// Mitsubishi GX Works2 project: PLC_Group_12   PLC: FX3G

// global labels: Global1
VAR_GLOBAL
  start_day AT X010 : BOOL;
  flour_input AT D1100 : REAL;
  yeast_input AT D1102 : REAL;
  water_input AT D1104 : REAL;
  oil_input AT D1106 : REAL;
  spices_input AT D1108 : REAL;
  flour_stock AT D1110 : REAL;
  yeast_stock AT D1112 : REAL;
  water_stock AT D1114 : REAL;
  oil_stock AT D1116 : REAL;
  spices_stock AT D1118 : REAL;
  input AT M0 : BOOL;
END_VAR
VAR_GLOBAL CONSTANT
  min_flour : REAL := 100;
END_VAR
VAR_GLOBAL
  enough_flour AT M20 : BOOL;
  const1 AT E5.0 : REAL;
  const2 AT E2.0 : REAL;
  const4 AT E10.0 : REAL;
  const3 AT E0.3 : REAL;
  enough_yeast AT M40 : BOOL;
  enough_water AT M42 : BOOL;
  enough_oil AT M44 : BOOL;
  enough_spices AT M46 : BOOL;
  emergemcy_stop AT X007 : BOOL;
  all_ok AT M6 : BOOL;
  can_start AT M52 : BOOL;
  in_process AT Y010 : BOOL;
  flour_tank AT D1120 : REAL;
  yeast_tank AT D1122 : REAL;
  water_tank AT D1124 : REAL;
  oil_tank AT D1126 : REAL;
  spices_tank AT D1128 : REAL;
  start_prepare AT X002 : BOOL;
  sub_flour AT E100 : REAL;
  add_flour AT E100 : REAL;
  sub_yeast AT E20 : REAL;
  add_yeast AT E20 : REAL;
  sub_water AT E50 : REAL;
  add_water AT E50 : REAL;
  sub_oil AT E30 : REAL;
  add_oil AT E30 : REAL;
  sub_spices AT E10 : REAL;
  add_spices AT E10 : REAL;
  preparing_lamp AT Y005 : BOOL;
  preparing_timer AT TC200 : BOOL;
  timer_stopped AT TS200 : BOOL;
  start_mix AT X001 : BOOL;
  mix_tank AT D1130 : REAL;
  rst_flour AT E0.0 : REAL;
  rst_material AT E0.0 : REAL;
  mixTankActivaited AT M101 : BOOL;
  mixer_lamp AT Y001 : BOOL;
  start_swelling AT X011 : BOOL;
  counter_one AT CC0 : BOOL;
  swelling_tank AT D1132 : REAL;
  counter AT CS0 : BOOL;
  swellingProccesActivated AT M102 : BOOL;
  swelling_timer AT TC201 : BOOL;
  one_sec_pulse AT M8013 : BOOL;
  swelling_one AT Y002 : BOOL;
  swelling_two AT Y003 : BOOL;
  timer_two_stopped AT TS201 : BOOL;
  baking_procces_activated AT M103 : BOOL;
  baking_pan AT D1134 : REAL;
  baking_timer AT TC202 : BOOL;
  baking_lamp AT Y004 : BOOL;
  quality_ck AT X003 : BOOL;
  quality AT D8281 : INT;
  temp_analog_value AT D1200 : INT;
  quality_value AT D1202 : REAL;
  qc_approve AT M104 : BOOL;
  qc_fail_counter AT CC2 : BOOL;
  qc_timer AT TC203 : BOOL;
  qc_lamp AT Y006 : BOOL;
  shelves AT D1136 : REAL;
  QA_Activated AT M105 : BOOL;
  all_reset AT M340 : BOOL;
  not_enough_material AT M341 : BOOL;
  TC204 : BOOL;
  end_timer AT TC204 : BOOL;
  stop_acticated AT M350 : BOOL;
  emptyMix_Tank_checkPulse : BOOL;
  day_active_counter AT CC8 : BOOL;
  preperingLampIsOver AT M110 : BOOL;
  moveToTanksConfimation AT M100 : BOOL;
  bakingLampsOver AT M112 : BOOL;
  stopSystemTimerActivated AT M342 : BOOL;
  test AT M106 : BOOL;
  testtwo AT M107 : BOOL;
  qc_approval AT M108 : BOOL;
  testthree AT M109 : BOOL;
END_VAR

// task Task_01 (event TRUE, interval 0, priority 31): POU_01

PROGRAM POU_01
VAR
  day_active : BOOL;
END_VAR
(* structured ladder/FBD written out as ST: instructions are called as NAME(EN, inputs, outputs); _pN, _eN, _tN stand for wires *)
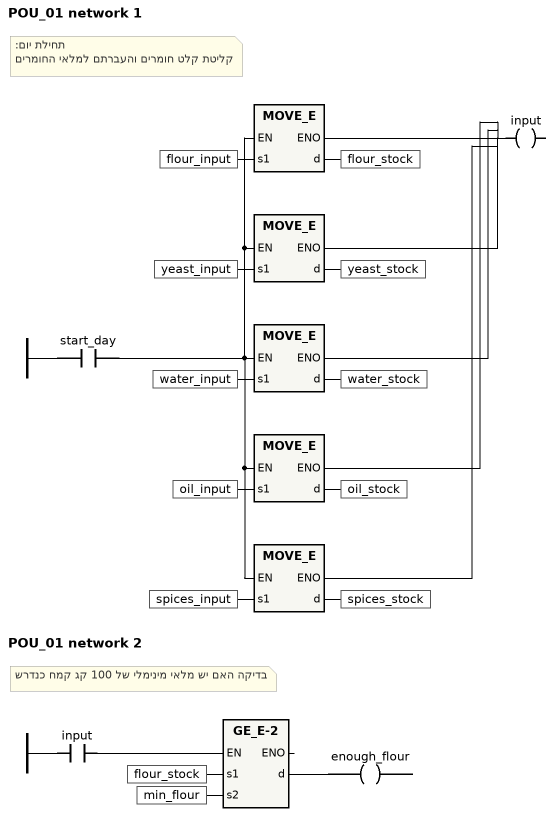
(* network 1 *)
(* תחילת יום: /  קליטת קלט חומרים והעברתם למלאי החומרים *)
_e1 := MOVE_E(start_day, flour_input, flour_stock);
_e2 := MOVE_E(start_day, yeast_input, yeast_stock);
_e3 := MOVE_E(start_day, water_input, water_stock);
_e4 := MOVE_E(start_day, oil_input, oil_stock);
_e5 := MOVE_E(start_day, spices_input, spices_stock);
input := _e1 OR _e2 OR _e3 OR _e4 OR _e5;
(* network 2 *)
(* בדיקה האם יש מלאי מינימלי של 100 קג קמח כנדרש *)
GE_E(input, flour_stock, min_flour, _t1);
enough_flour := _t1;
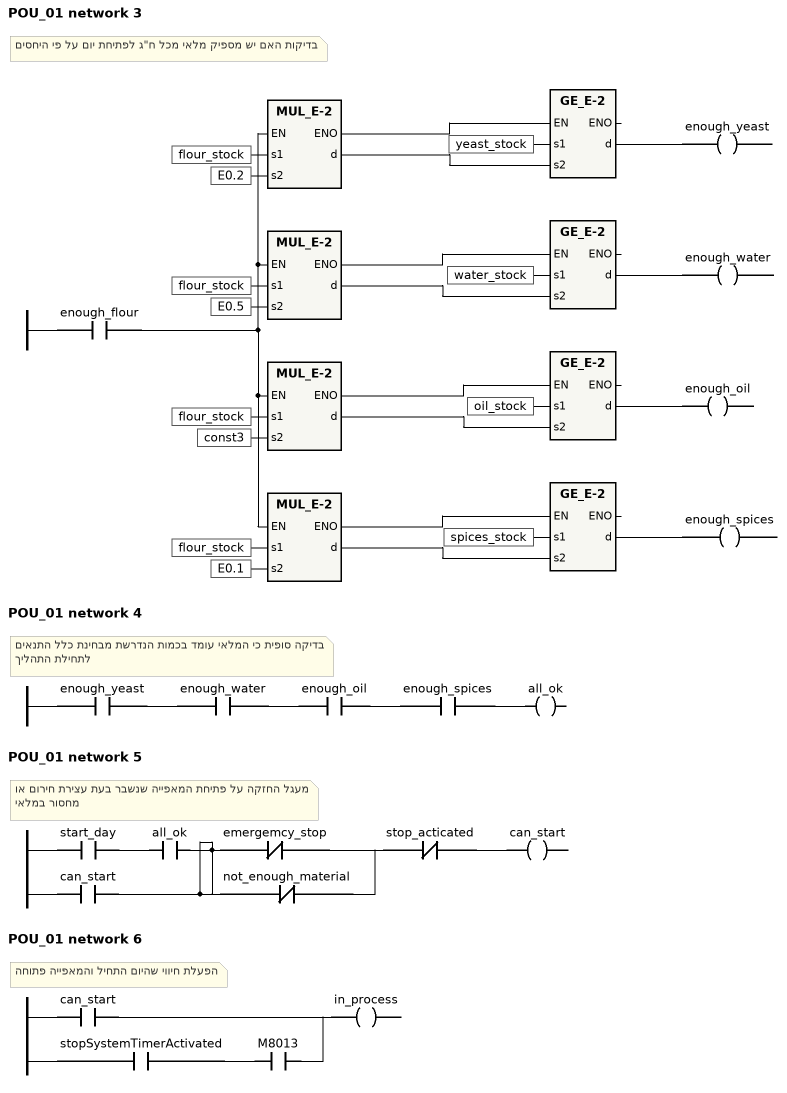
(* network 3 *)
(* בדיקות האם יש מספיק מלאי מכל ח"ג לפתיחת יום על פי היחסים *)
_e2 := MUL_E(enough_flour, flour_stock, E0.2, _t1);
GE_E(_e2, yeast_stock, _t1, _t3);
enough_yeast := _t3;
_e5 := MUL_E(enough_flour, flour_stock, E0.5, _t4);
GE_E(_e5, water_stock, _t4, _t6);
enough_water := _t6;
_e8 := MUL_E(enough_flour, flour_stock, const3, _t7);
GE_E(_e8, oil_stock, _t7, _t9);
enough_oil := _t9;
_e11 := MUL_E(enough_flour, flour_stock, E0.1, _t10);
GE_E(_e11, spices_stock, _t10, _t12);
enough_spices := _t12;
(* network 4 *)
(* בדיקה סופית כי המלאי עומד בכמות הנדרשת מבחינת כלל התנאים לתחילת התהליך *)
all_ok := enough_yeast AND enough_water AND enough_oil AND enough_spices;
(* network 5 *)
(* מעגל החזקה על פתיחת המאפייה שנשבר בעת עצירת חירום או מחסור במלאי *)
_p1 := (start_day AND all_ok) OR can_start;
can_start := ((_p1 AND NOT emergemcy_stop) OR (_p1 AND NOT not_enough_material)) AND NOT stop_acticated;
(* network 6 *)
(* הפעלת חיווי שהיום התחיל והמאפייה פתוחה *)
in_process := can_start OR (stopSystemTimerActivated AND M8013);
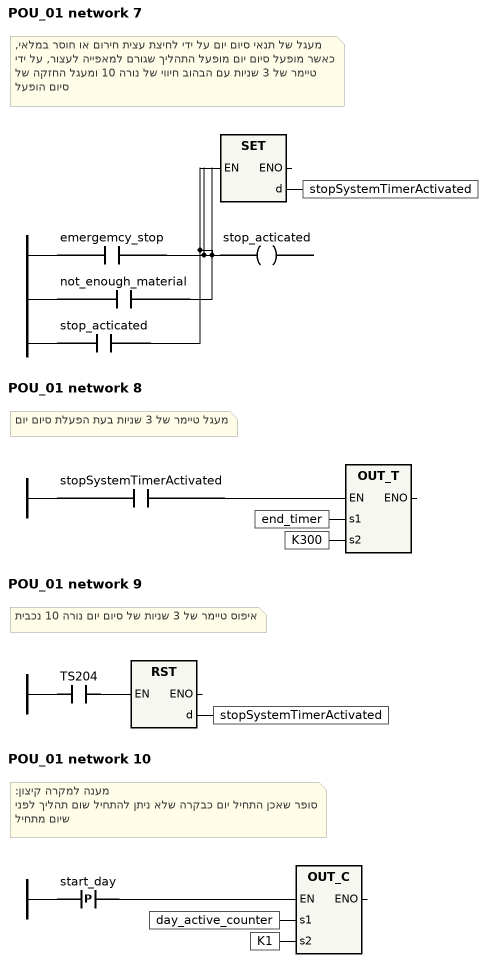
(* network 7 *)
(* מעגל של תנאי סיום יום על ידי לחיצת עצית חירום או חוסר במלאי, /  כאשר מופעל סיום יום מופעל התהליך שגורם למאפייה לעצור, על ידי טיימר של 3 שניות עם הבהוב חיווי של נורה 10 ומעגל החזקה של סיום הופעל *)
_p1 := emergemcy_stop OR not_enough_material OR stop_acticated;
SET(_p1, stopSystemTimerActivated);
stop_acticated := _p1;
(* network 8 *)
(* מעגל טיימר של 3 שניות בעת הפעלת סיום יום *)
OUT_T(stopSystemTimerActivated, end_timer, K300);
(* network 9 *)
(* איפוס טיימר של 3 שניות של סיום יום נורה 10 נכבית *)
RST(TS204, stopSystemTimerActivated);
(* network 10 *)
(* מענה למקרה קיצון: / סופר שאכן התחיל יום כבקרה שלא ניתן להתחיל שום תהליך לפני שיום מתחיל *)
OUT_C(LDP(TRUE, start_day), day_active_counter, K1);
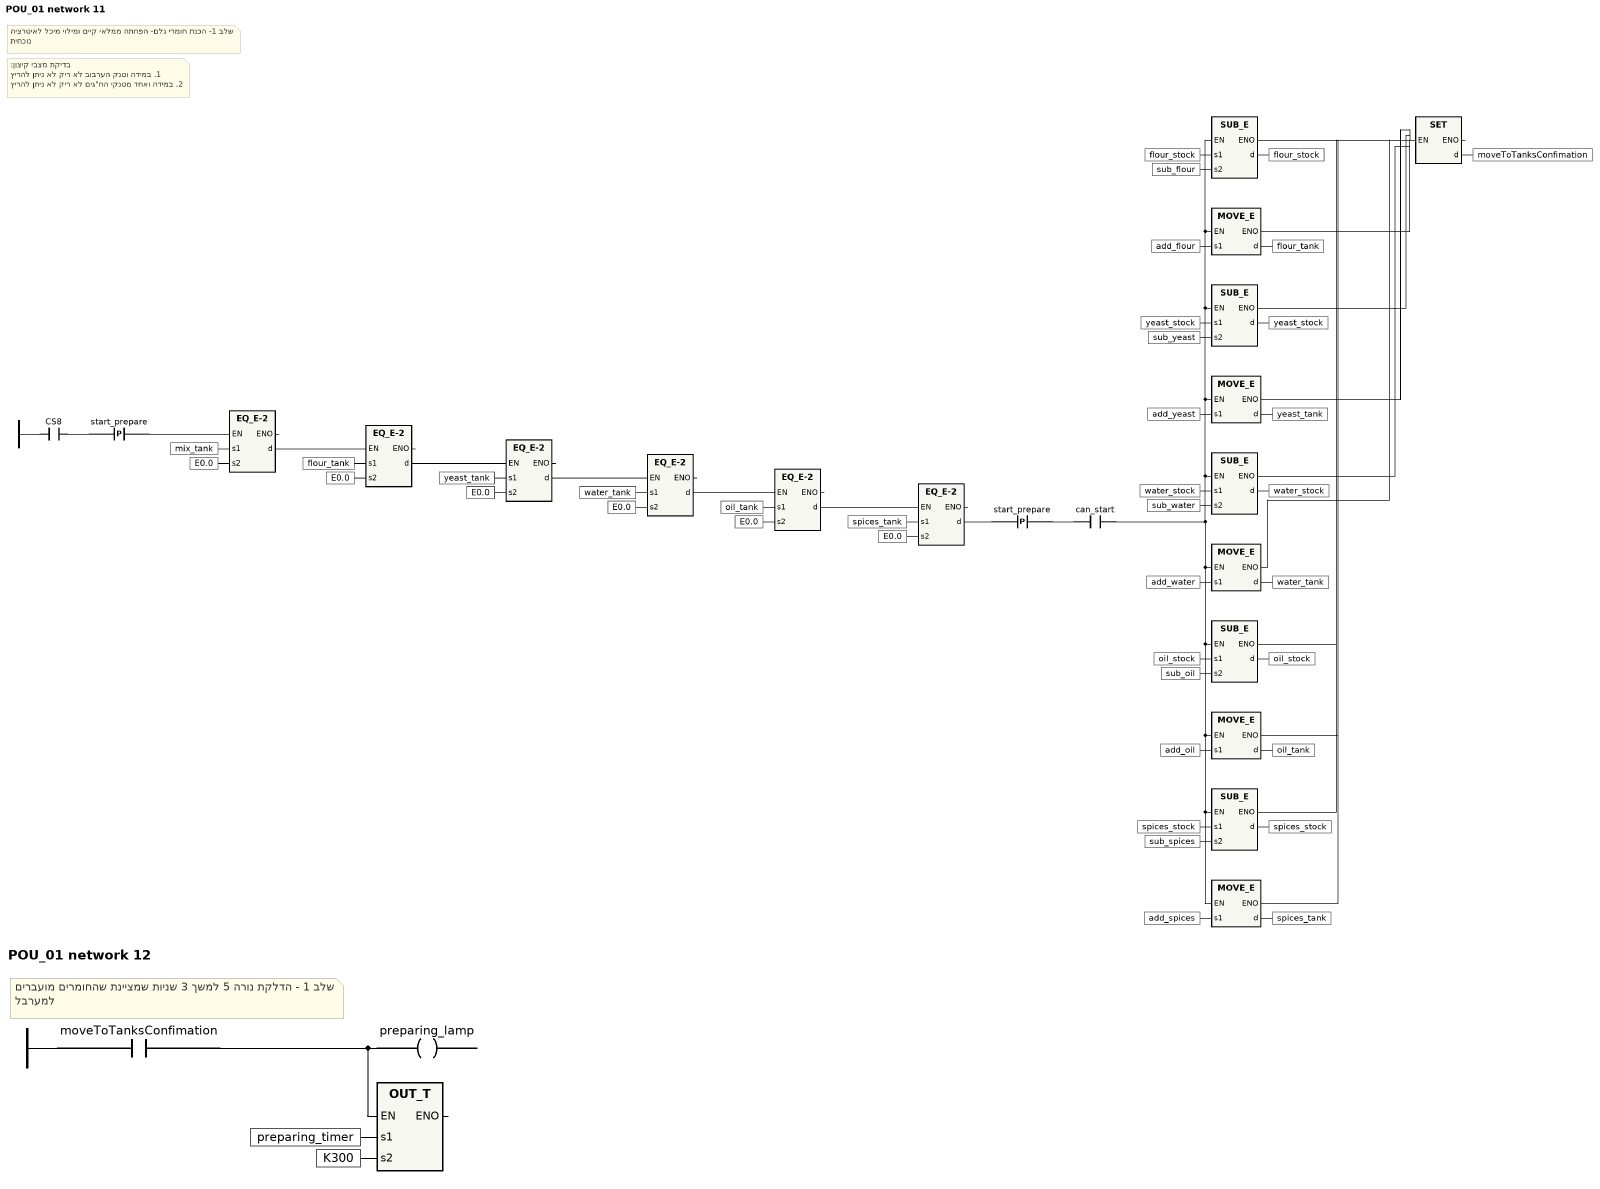
(* network 11 *)
(* שלב 1- הכנת חומרי גלם- הפחתה ממלאי קיים ומילוי מיכל לאיטרציה נוכחית *)
(* בדיקת מצבי קיצון: / 1. במידה וטנק הערבוב לא ריק לא ניתן להריץ / 2. במידה ואחד מטנקי הח"גים לא ריק לא ניתן להריץ *)
EQ_E(CS8 AND LDP(TRUE, start_prepare), mix_tank, E0.0, _t1);
EQ_E(_t1, flour_tank, E0.0, _t2);
EQ_E(_t2, yeast_tank, E0.0, _t3);
EQ_E(_t3, water_tank, E0.0, _t4);
EQ_E(_t4, oil_tank, E0.0, _t5);
EQ_E(_t5, spices_tank, E0.0, _t6);
_p7 := _t6 AND LDP(TRUE, start_prepare) AND can_start;
_e8 := SUB_E(_p7, flour_stock, sub_flour, flour_stock);
_e9 := MOVE_E(_p7, add_flour, flour_tank);
_e10 := SUB_E(_p7, yeast_stock, sub_yeast, yeast_stock);
_e11 := MOVE_E(_p7, add_yeast, yeast_tank);
_e12 := SUB_E(_p7, water_stock, sub_water, water_stock);
_e13 := MOVE_E(_p7, add_water, water_tank);
_e14 := SUB_E(_p7, oil_stock, sub_oil, oil_stock);
_e15 := MOVE_E(_p7, add_oil, oil_tank);
_e16 := SUB_E(_p7, spices_stock, sub_spices, spices_stock);
_e17 := MOVE_E(_p7, add_spices, spices_tank);
SET(_e8 OR _e9 OR _e10 OR _e11 OR _e12 OR _e13 OR _e14 OR _e15 OR _e16 OR _e17, moveToTanksConfimation);
(* network 12 *)
(* שלב 1 - הדלקת נורה 5 למשך 3 שניות שמציינת שהחומרים מועברים למערבל *)
preparing_lamp := moveToTanksConfimation;
OUT_T(moveToTanksConfimation, preparing_timer, K300);
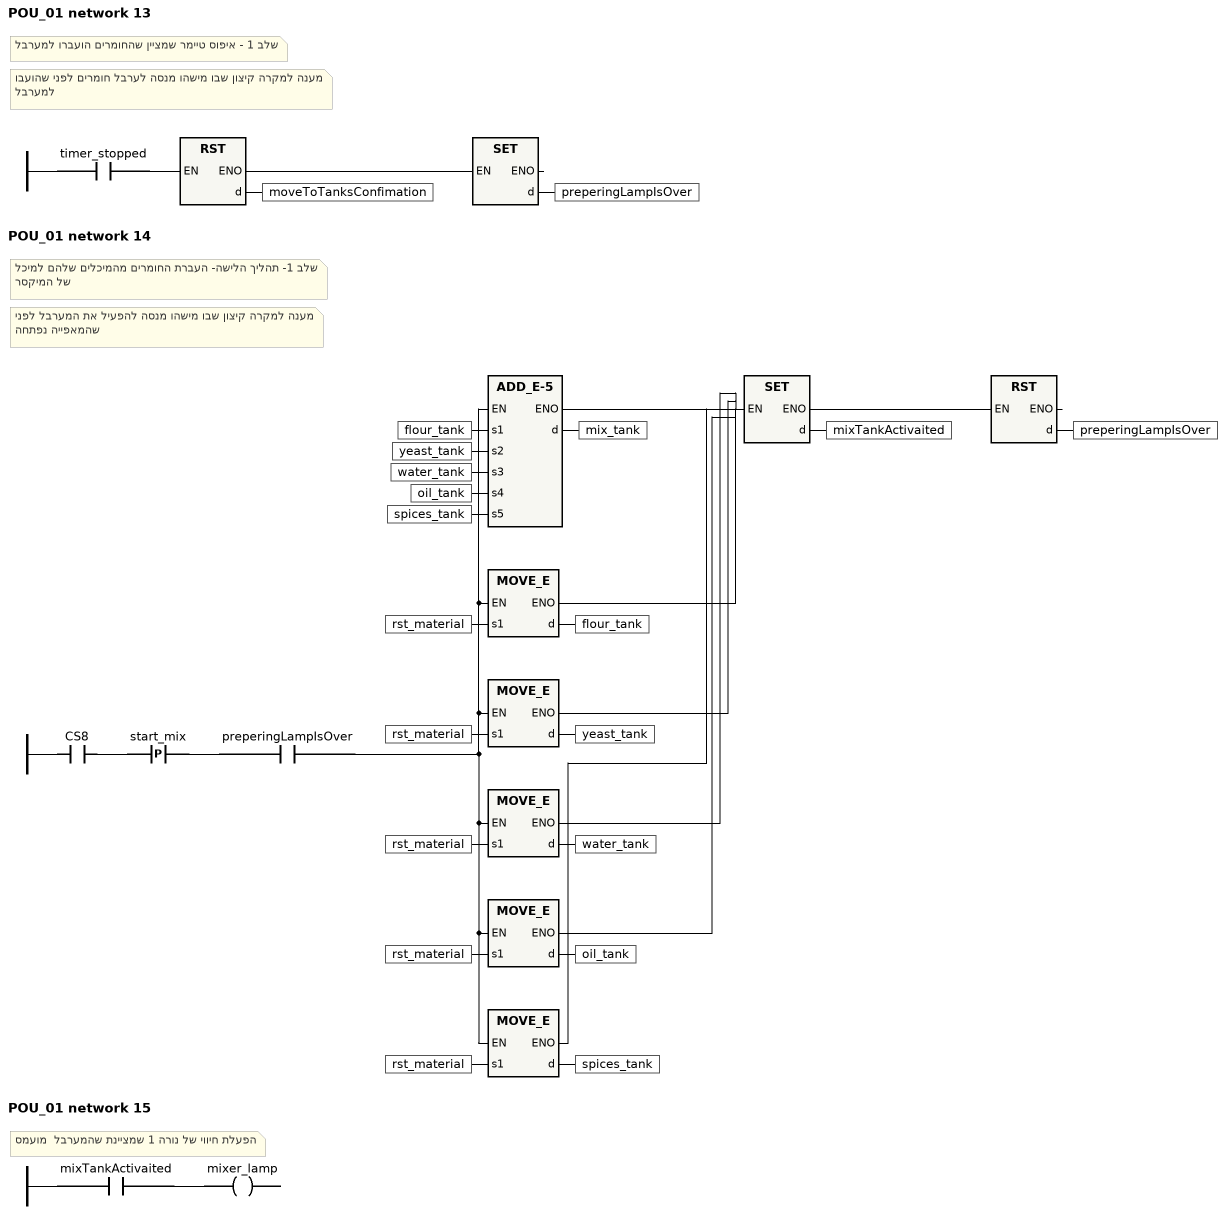
(* network 13 *)
(* שלב 1 - איפוס טיימר שמציין שהחומרים הועברו למערבל *)
(* מענה למקרה קיצון שבו מישהו מנסה לערבל חומרים לפני שהועבו למערבל *)
_e1 := RST(timer_stopped, moveToTanksConfimation);
SET(_e1, preperingLampIsOver);
(* network 14 *)
(* שלב 1- תהליך הלישה- העברת החומרים מהמיכלים שלהם למיכל של המיקסר *)
(* מענה למקרה קיצון שבו מישהו מנסה להפעיל את המערבל לפני שהמאפייה נפתחה *)
_p1 := CS8 AND LDP(TRUE, start_mix) AND preperingLampIsOver;
_e2 := ADD_E(_p1, flour_tank, yeast_tank, water_tank, oil_tank, spices_tank, mix_tank);
_e3 := MOVE_E(_p1, rst_material, flour_tank);
_e4 := MOVE_E(_p1, rst_material, yeast_tank);
_e5 := MOVE_E(_p1, rst_material, water_tank);
_e6 := MOVE_E(_p1, rst_material, oil_tank);
_e7 := MOVE_E(_p1, rst_material, spices_tank);
_e8 := SET(_e2 OR _e3 OR _e4 OR _e5 OR _e6 OR _e7, mixTankActivaited);
RST(_e8, preperingLampIsOver);
(* network 15 *)
(* הפעלת חיווי של נורה 1 שמציינת שהמערבל  מועמס *)
mixer_lamp := mixTankActivaited;
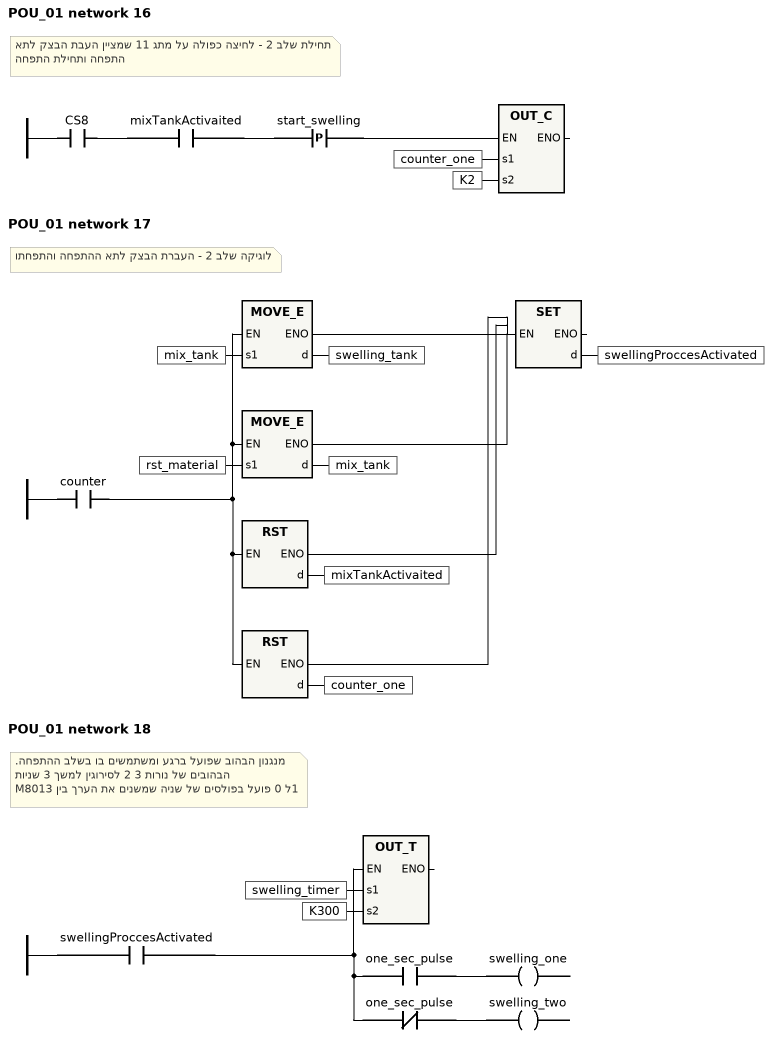
(* network 16 *)
(* תחילת שלב 2 - לחיצה כפולה על מתג 11 שמציין העבת הבצק לתא התפחה ותחילת התפחה *)
OUT_C(CS8 AND mixTankActivaited AND LDP(TRUE, start_swelling), counter_one, K2);
(* network 17 *)
(* לוגיקה שלב 2 - העברת הבצק לתא ההתפחה והתפחתו *)
_e1 := MOVE_E(counter, mix_tank, swelling_tank);
_e2 := MOVE_E(counter, rst_material, mix_tank);
_e3 := RST(counter, mixTankActivaited);
_e4 := RST(counter, counter_one);
SET(_e1 OR _e2 OR _e3 OR _e4, swellingProccesActivated);
(* network 18 *)
(* מנגנון הבהוב שפועל ברגע ומשתמשים בו בשלב ההתפחה. / הבהובים של נורות 2 3 לסירוגין למשך 3 שניות /  / M8013 פועל בפולסים של שניה שמשנים את הערך בין 0 ל1 *)
OUT_T(swellingProccesActivated, swelling_timer, K300);
swelling_one := swellingProccesActivated AND one_sec_pulse;
swelling_two := swellingProccesActivated AND NOT one_sec_pulse;
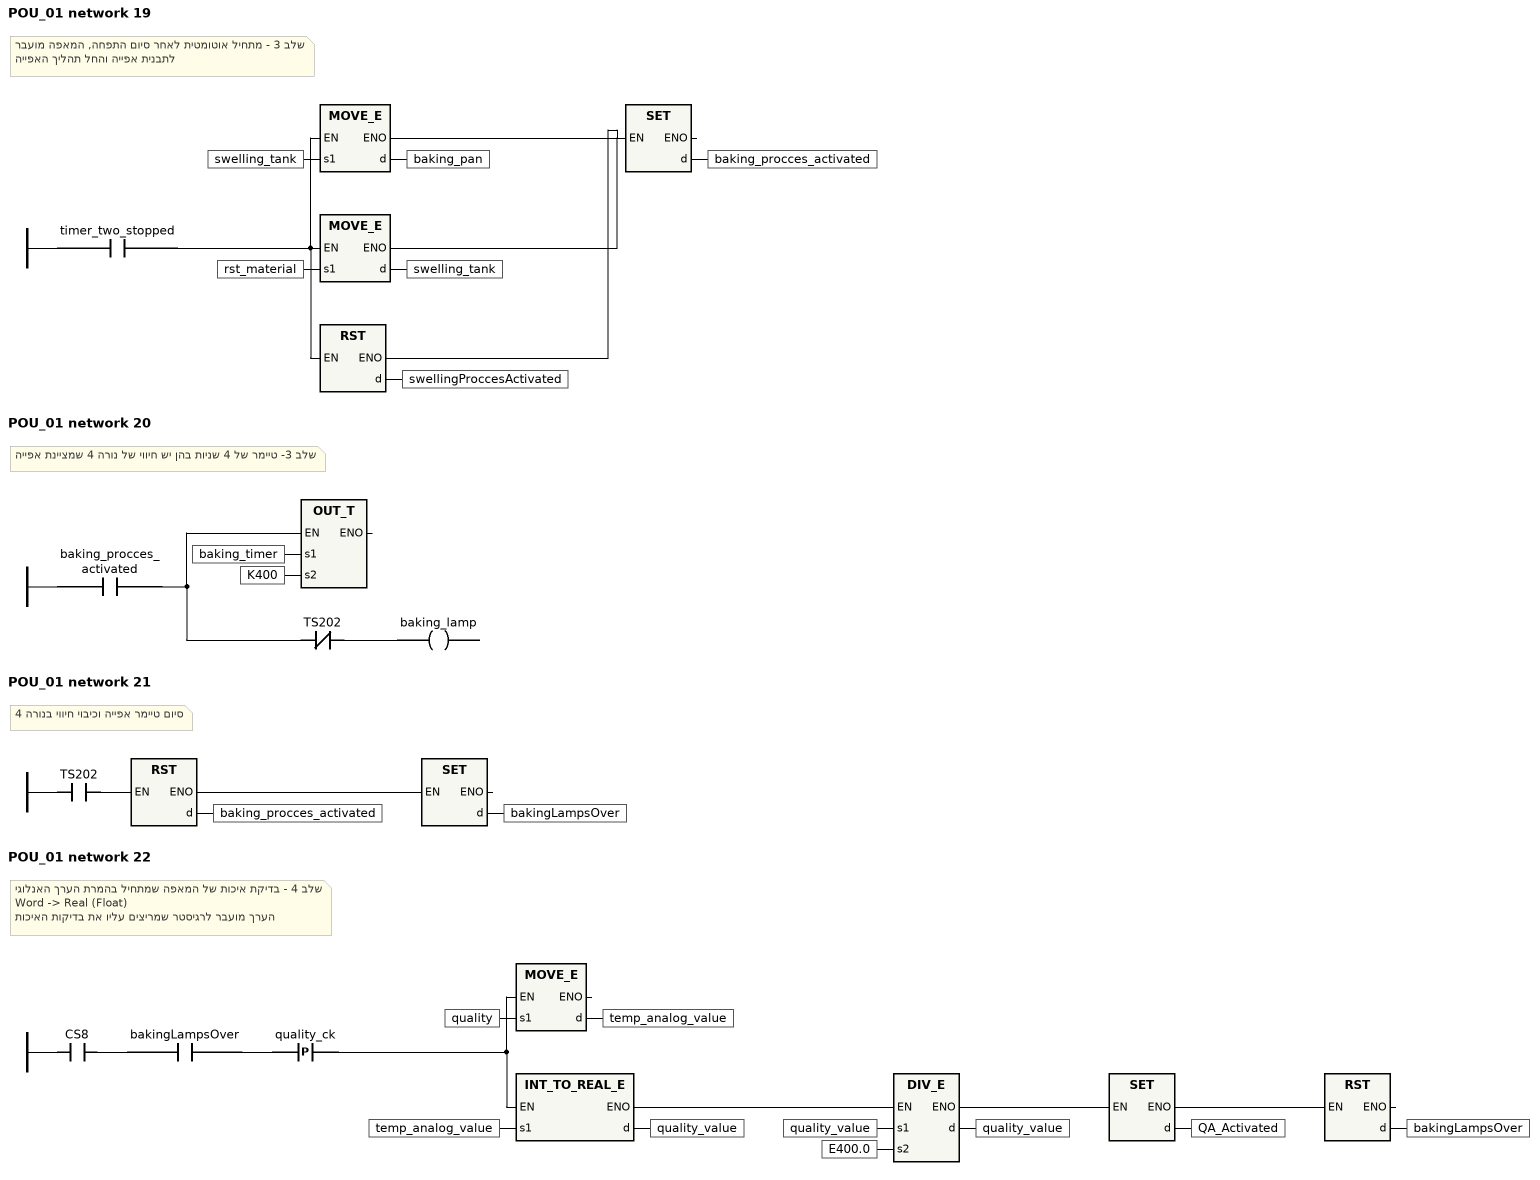
(* network 19 *)
(* שלב 3 - מתחיל אוטומטית לאחר סיום התפחה, המאפה מועבר לתבנית אפייה והחל תהליך האפייה *)
_e1 := MOVE_E(timer_two_stopped, swelling_tank, baking_pan);
_e2 := MOVE_E(timer_two_stopped, rst_material, swelling_tank);
_e3 := RST(timer_two_stopped, swellingProccesActivated);
SET(_e1 OR _e2 OR _e3, baking_procces_activated);
(* network 20 *)
(* שלב 3- טיימר של 4 שניות בהן יש חיווי של נורה 4 שמציינת אפייה *)
OUT_T(baking_procces_activated, baking_timer, K400);
baking_lamp := baking_procces_activated AND NOT TS202;
(* network 21 *)
(* סיום טיימר אפייה וכיבוי חיווי בנורה 4 *)
_e1 := RST(TS202, baking_procces_activated);
SET(_e1, bakingLampsOver);
(* network 22 *)
(* שלב 4 - בדיקת איכות של המאפה שמתחיל בהמרת הערך האנלוגי  / Word -> Real (Float) / הערך מועבר לרגיסטר שמריצים עליו את בדיקות האיכות *)
_p1 := CS8 AND bakingLampsOver AND LDP(TRUE, quality_ck);
MOVE_E(_p1, quality, temp_analog_value);
_e2 := INT_TO_REAL_E(_p1, temp_analog_value, quality_value);
_e3 := DIV_E(_e2, quality_value, E400.0, quality_value);
_e4 := SET(_e3, QA_Activated);
RST(_e4, bakingLampsOver);
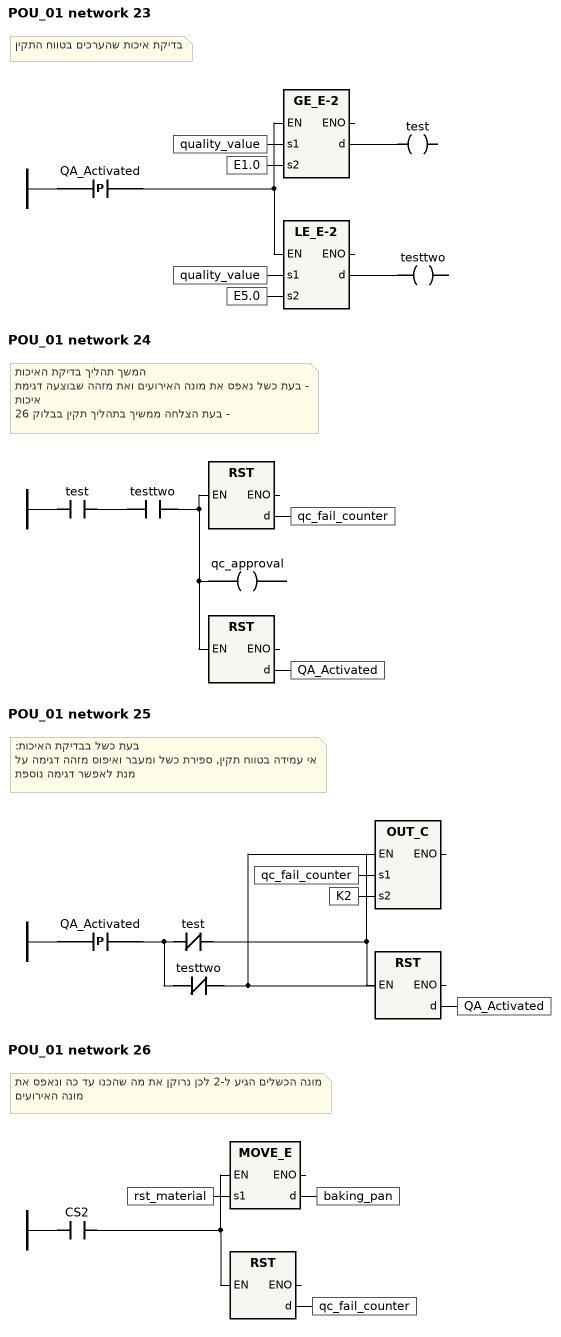
(* network 23 *)
(* בדיקת איכות שהערכים בטווח התקין *)
_p1 := LDP(TRUE, QA_Activated);
GE_E(_p1, quality_value, E1.0, _t2);
test := _t2;
LE_E(_p1, quality_value, E5.0, _t3);
testtwo := _t3;
(* network 24 *)
(* המשך תהליך בדיקת האיכות  / - בעת כשל נאפס את מונה האירועים ואת מזהה שבוצעה דגימת איכות / - בעת הצלחה ממשיך בתהליך תקין בבלוק 26 *)
_p1 := test AND testtwo;
qc_approval := _p1;
RST(_p1, qc_fail_counter);
RST(_p1, QA_Activated);
(* network 25 *)
(* בעת כשל בבדיקת האיכות: / אי עמידה בטווח תקין, ספירת כשל ומעבר ואיפוס מזהה דגימה על מנת לאפשר דגימה נוספת *)
_p1 := LDP(TRUE, QA_Activated);
_p2 := (_p1 AND NOT test) OR (_p1 AND NOT testtwo);
OUT_C(_p2, qc_fail_counter, K2);
RST(_p2, QA_Activated);
(* network 26 *)
(* מונה הכשלים הגיע ל-2 לכן נרוקן את מה שהכנו עד כה ונאפס את מונה האירועים *)
MOVE_E(CS2, rst_material, baking_pan);
RST(CS2, qc_fail_counter);
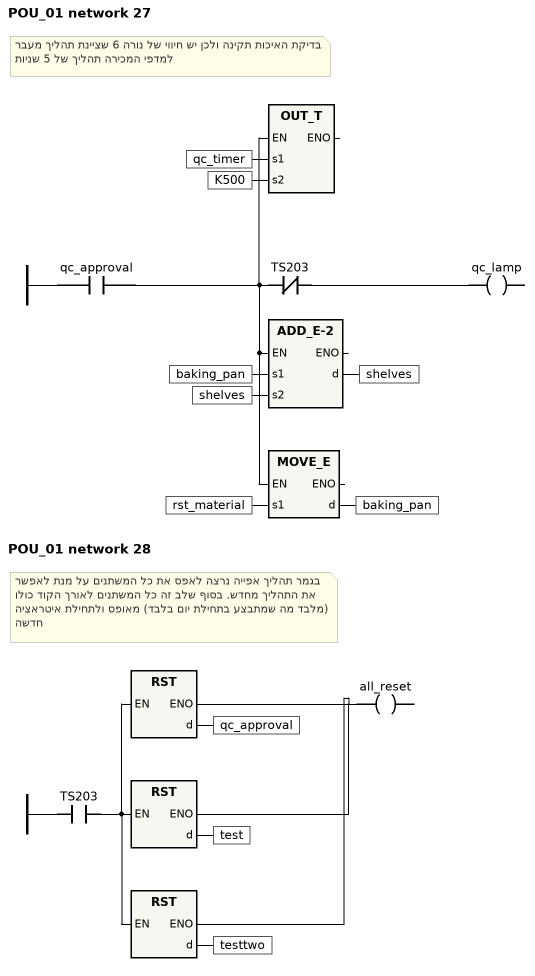
(* network 27 *)
(* בדיקת האיכות תקינה ולכן יש חיווי של נורה 6 שציינת תהליך מעבר למדפי המכירה תהליך של 5 שניות *)
OUT_T(qc_approval, qc_timer, K500);
qc_lamp := qc_approval AND NOT TS203;
ADD_E(qc_approval, baking_pan, shelves, shelves);
MOVE_E(qc_approval, rst_material, baking_pan);
(* network 28 *)
(* בגמר תהליך אפייה נרצה לאפס את כל המשתנים על מנת לאפשר את התהליך מחדש. בסוף שלב זה כל המשתנים לאורך הקוד כולו (מלבד מה שמתבצע בתחילת יום בלבד) מאופס ולתחילת איטראציה חדשה *)
_e1 := RST(TS203, qc_approval);
_e2 := RST(TS203, test);
_e3 := RST(TS203, testtwo);
all_reset := _e1 OR _e2 OR _e3;
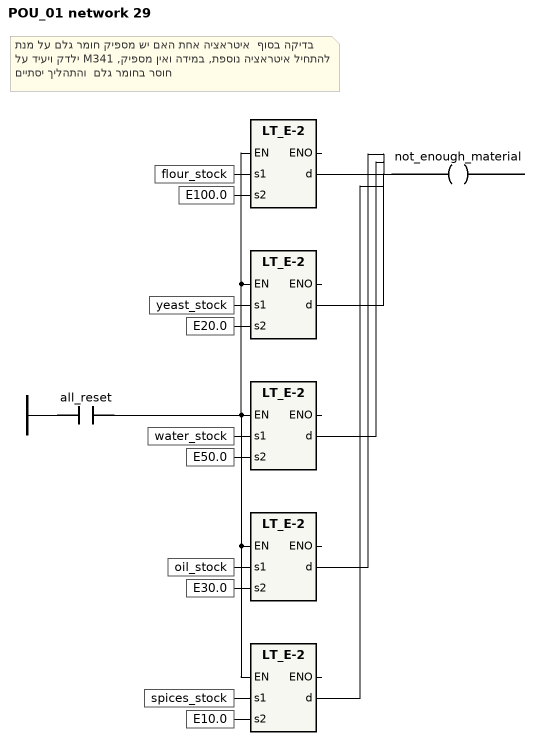
(* network 29 *)
(* בדיקה בסוף  איטראציה אחת האם יש מספיק חומר גלם על מנת להתחיל איטראציה נוספת, במידה ואין מספיק, M341 ילדק ויעיד על חוסר בחומר גלם  והתהליך יסתיים *)
LT_E(all_reset, flour_stock, E100.0, _t1);
LT_E(all_reset, yeast_stock, E20.0, _t2);
LT_E(all_reset, water_stock, E50.0, _t3);
LT_E(all_reset, oil_stock, E30.0, _t4);
LT_E(all_reset, spices_stock, E10.0, _t5);
not_enough_material := _t1 OR _t2 OR _t3 OR _t4 OR _t5;
END_PROGRAM
